FUNCTION_BLOCK X2Y2_J2 (* Compute X^2-Y^2 in Java without ECC *)
  (* Standard: 61499-1 *)
  (* Version 0.0, 2003-08-13, JHC, Rockwell Automation, Derived from X2Y2_J *)
  (* Compiler header: package fb.rt.student; import fb.rt.math.*; *)
  (* Compiler Java IBM Jikes 1.0.6 *)
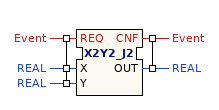
  EVENT_INPUT
    REQ WITH X, Y;
  END_EVENT
  EVENT_OUTPUT
    CNF WITH OUT;
  END_EVENT
  VAR_INPUT
    X : REAL;
    Y : REAL;
  END_VAR
  VAR_OUTPUT
    OUT : REAL;
  END_VAR
  ALGORITHM REQ IN Java:
OUT.value = (X.value-Y.value)*(X.value+Y.value);
CNF.serviceEvent(this);
  END_ALGORITHM
END_FUNCTION_BLOCK
